(* CoDeSys 2.3.9.37 project: Cap9_1.pro *)
(* Libraries: Standard.LIB 4.10.05 12:14:46 *)

(* Global variable list: Global_Variables *)
VAR_GLOBAL

(* Variables de entrada *)
    Numero: INT ;


(* Variables de Salida*)
      a0:BOOL;
	b0:BOOL;
	c0:BOOL;
	d0:BOOL;
	e0:BOOL;
	f0:BOOL;
	g0:BOOL;
      Novalido:BOOL;

END_VAR

(* POU PLC_PRG, ST *)
PROGRAM PLC_PRG
VAR
END_VAR

END_PROGRAM

(* Visualisation Display
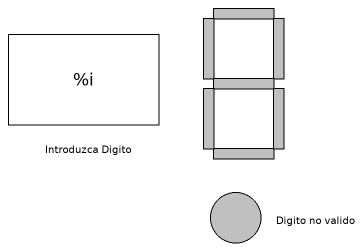
rectangle at (265,64)-(326,75): alarm colour if a0
rectangle at (325,74)-(336,135): alarm colour if b0
rectangle at (255,74)-(266,135): alarm colour if f0
rectangle at (265,134)-(326,145): alarm colour if g0
rectangle at (265,204)-(326,215): alarm colour if d0
rectangle at (325,144)-(336,205): alarm colour if c0
rectangle at (255,144)-(266,205): alarm colour if e0
rectangle at (60,90)-(211,181): text "%i"; shows Numero; editable
ellipse at (262,248)-(313,299): alarm colour if Novalido
rectangle at (60,190)-(221,221): text "Introduzca Digito"
rectangle at (287,261)-(448,292): text "Digito no valido"
*)
